// Mitsubishi GX Works2 project: 步进电机自动速度7速   PLC: FX3U/FX3UC

PROGRAM MAIN
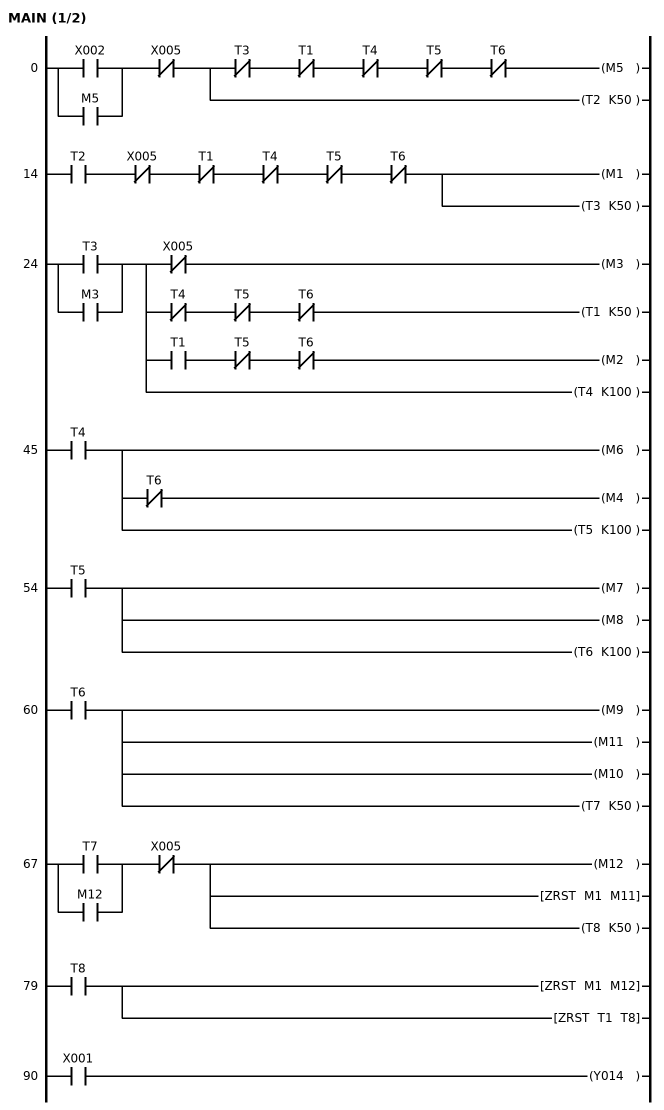
0     LD      X002
      OR      M5
      ANI     X005
      MPS
      ANI     T3
      ANI     T1
      ANI     T4
      ANI     T5
      ANI     T6
      OUT     M5
      MPP
      OUT     T2 K50
14    LD      T2
      ANI     X005
      ANI     T1
      ANI     T4
      ANI     T5
      ANI     T6
      OUT     M1
      OUT     T3 K50
24    LD      T3
      OR      M3
      MPS
      ANI     X005
      OUT     M3
      MRD
      ANI     T4
      ANI     T5
      ANI     T6
      OUT     T1 K50
      MRD
      AND     T1
      ANI     T5
      ANI     T6
      OUT     M2
      MPP
      OUT     T4 K100
45    LD      T4
      OUT     M6
      MPS
      ANI     T6
      OUT     M4
      MPP
      OUT     T5 K100
54    LD      T5
      OUT     M7
      OUT     M8
      OUT     T6 K100
60    LD      T6
      OUT     M9
      OUT     M11
      OUT     M10
      OUT     T7 K50
67    LD      T7
      OR      M12
      ANI     X005
      OUT     M12
      ZRST    M1 M11
      OUT     T8 K50
79    LD      T8
      ZRST    M1 M12
      ZRST    T1 T8
90    LD      X001
      OUT     Y014
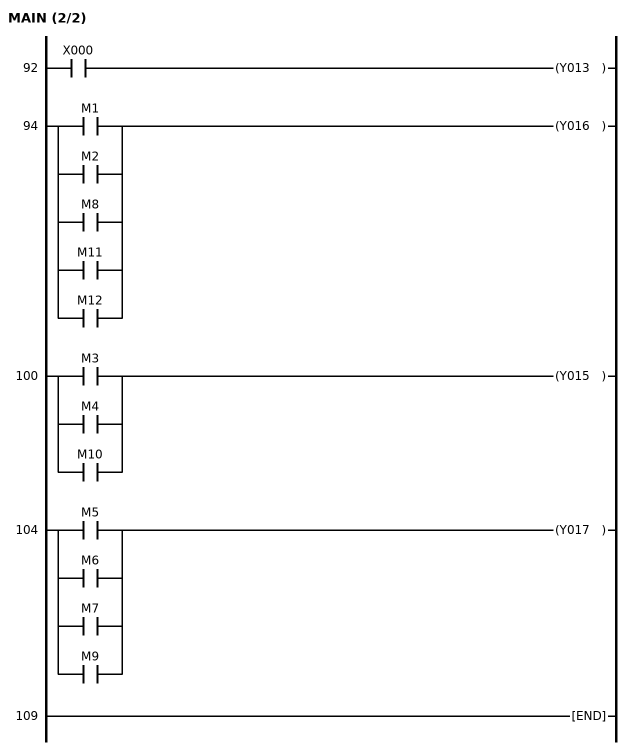
92    LD      X000
      OUT     Y013
94    LD      M1
      OR      M2
      OR      M8
      OR      M11
      OR      M12
      OUT     Y016
100   LD      M3
      OR      M4
      OR      M10
      OUT     Y015
104   LD      M5
      OR      M6
      OR      M7
      OR      M9
      OUT     Y017
109   END
END_PROGRAM
